// TIA Portal project "MILL" (V18)

(* hardware
DEVICE "S7-1200-Station_1"  S7-1200 Station
   slot 0: "Baugruppenträger_0"  S7-1200 Rack  Rack  V1.0
   slot 1: "MILL"  CPU 1215C DC/DC/DC  6ES7 215-1AG40-0XB0  V4.5
*)

// ===== PLC "MILL"  CPU 1215C DC/DC/DC =====

VAR_GLOBAL   // PLC tag table "Variablentabelle_1"
   "band_rein" AT %Q0.0 : Bool;   // DQa.0
   "eingang_LS" AT %I0.0 : Bool;   // DIa.0
   "bearbeitung_LS" AT %I0.1 : Bool;   // DIa.1
   "sauger_innen" AT %I0.2 : Bool;   // DIa.2
   "sauger_außen" AT %I0.3 : Bool;   // DIa.3
   "band_raus" AT %Q0.1 : Bool;   // DQa.1
   "sauger_rein" AT %Q0.2 : Bool;   // DQa.2
   "sauger_raus" AT %Q0.3 : Bool;   // DQa.3
   "sauger_unten" AT %Q0.4 : Bool;   // DQa.4
   "ventil_vakuum" AT %Q0.5 : Bool;   // DQa.5
   "kompressor" AT %Q0.6 : Bool;   // DQa.6
   "fraese" AT %Q0.7 : Bool;   // DQa.7
   "band_PWM" AT %Q1.0 : Bool;   // DQb.0
   "sauger_PWM" AT %Q1.1 : Bool;   // DQb.1
END_VAR

DATA_BLOCK "LOOP_DB"   // DB1
{ S7_Optimized_Access := 'TRUE' }
VERSION : 0.1
// stored: InstanceOfName LOOP
"LOOP"
BEGIN
END_DATA_BLOCK

FUNCTION_BLOCK "LOOP"   // FB1, SCL
{ S7_Optimized_Access := 'TRUE' }
VERSION : 0.1
   VAR
      warte : TON_TIME;
      warte_zeit : Time := T#500ms;
      warte_start : Bool;
      "step" : Int;
      pick : Bool;
      drop : Bool;
      mill : Bool;
      pick_finished : Bool;
      drop_finished : Bool;
      mill_finished : Bool;
      duration : Int := 2;
      idle : Bool;
   END_VAR
   VAR RETAIN
      modell : String := 'MILL';
   END_VAR
   VAR
      pick_failed : Bool;
      drop_failed : Bool;
      drop_aktiv : Bool;
      pick_aktiv : Bool;
      mill_aktiv : Bool;
   END_VAR
   VAR RETAIN
      zeit_prozessende : Time := T#2000MS;
      zeit_vakuumloesen : Time := T#200MS;
      zeit_saugerRunter : Time := T#700MS;
      zeit_vorFehlercheck : Time := T#2S;
   END_VAR
   VAR
      zeit_FraesPause : Time := T#1S;
   END_VAR
   VAR RETAIN
      "version" : String := '1.0';
   END_VAR
BEGIN
   #warte(IN:=#warte_start,
               PT:=#warte_zeit);

   // Stepchain MILL
   CASE #step OF
       0: // init
           #step := 1;
       1: // rdy
           #idle := TRUE;
           #pick_finished := FALSE;
           #pick_failed := FALSE;
           #drop_finished := FALSE;
           #drop_failed := FALSE;
           #mill_finished := FALSE;
           #step := 5;
       5: // Fallunterscheidung
           IF #pick THEN
               #pick_aktiv := TRUE;
               #pick := FALSE;
               #idle := FALSE;
               #step := 10;
           ELSIF #drop THEN
               #drop_aktiv := TRUE;
               #drop := FALSE;
               #idle := FALSE;
               #step := 100;
           ELSIF #mill THEN
               #mill_aktiv := TRUE;
               #mill := FALSE;
               #idle := FALSE;
               #step := 40;
           END_IF;

       200: // Ende jedes Prozesses
           "ventil_vakuum" := FALSE;
           "band_PWM" := FALSE;
           "band_raus" := FALSE;
           "band_rein" := FALSE;
           "sauger_PWM" := FALSE;
           "sauger_raus" := FALSE;
           "sauger_rein" := FALSE;
           #warte_zeit := #zeit_prozessende;
           #warte_start := TRUE;
           IF #warte.Q THEN
               #warte_start := FALSE;
               #step := 1;
           END_IF
           ;
       10: // ----------------------------------------------------- START PICK
           // sauger raus bis schalter
           "sauger_PWM" := TRUE;
           "sauger_raus":= TRUE;
           IF "sauger_außen" THEN
               "sauger_raus" := FALSE;
               #step := 20;
           END_IF;
       20: // kurz warten
           #warte_zeit := T#200ms;
           #warte_start := TRUE;
           IF #warte.Q THEN
               #warte_start := FALSE;
               #step := 21;
           END_IF;
       21: // Sauger nimmt WP auf
           "kompressor" := TRUE;
           #step := 25;
       25: // warten
           #warte_zeit := T#200ms;
           #warte_start := TRUE;
           IF #warte.Q THEN
               #warte_start := FALSE;
               #step := 22;
           END_IF;
       22: // saugerkopf nach unten
           "sauger_unten" := TRUE;
           #step := 23;
       23: // Saugerkopf aktivieren
           #warte_zeit := #zeit_saugerRunter;
           #warte_start := TRUE;
           IF #warte.Q THEN
               "ventil_vakuum" := TRUE;
               #warte_start := FALSE;
               #step := 24;
           END_IF;
       24: // saugerkopf nach oben
           #warte_zeit := T#200ms;
           #warte_start := TRUE;
           IF #warte.Q THEN
               #warte_start := FALSE;
               "sauger_unten" := FALSE;
               #step := 30;
           END_IF
           ;
       30: // Sauger fährt rein
           "sauger_rein" := TRUE;
           IF "sauger_innen" THEN
               "sauger_rein" := FALSE;
               #step := 31;
           END_IF;
       31: // saugerkopf deaktivieren
           "sauger_unten" := TRUE;
           #warte_start := TRUE;
           #warte_zeit := #zeit_saugerRunter;
           IF #warte.Q THEN
               "ventil_vakuum" := FALSE;
               #warte_start := FALSE;
               #step := 32;
           END_IF;
       32: // kompressor aus
           #warte_start := TRUE;
           #warte_zeit := #zeit_vakuumloesen;
           IF #warte.Q THEN
               "kompressor" := FALSE;
               #warte_start := FALSE;
               #step := 33;
           END_IF;
       33: // saugerkopf nach oben und aus
           "sauger_unten" := FALSE;
           #warte_start := TRUE;
           #warte_zeit := #zeit_vorFehlercheck;
           IF #warte.Q THEN
               #warte_start := FALSE;
               #step := 34;
           END_IF;
       34: // warten und fertig
           IF "eingang_LS" THEN // Fehlercheck
               #pick_failed := TRUE;
           ELSE
               #pick_finished := TRUE;
           END_IF;
           #pick_aktiv := FALSE;
           #step := 200;
               // ------------------------- END PICK
       40: // ----------------------------------------------------- START MILL
           // Power auf Band
           "band_PWM" := TRUE;
           #step := 41;
       41: // band rein wenn LS 
           "band_rein" := TRUE;
           IF NOT "bearbeitung_LS" THEN
               #step := 42;
           END_IF;
       42: // Band laufen lassen bis mittig über Fräse
           #warte_start := TRUE;
           #warte_zeit := T#200ms;
           IF #warte.Q THEN
               "band_rein" := FALSE;
               #warte_start := FALSE;
               #step := 43;
           END_IF;

           // ----------------------------------------------------------------------- AufgabenLösung
           // 
       43: // Fräsen
           "fraese" := TRUE;
           #warte_start := TRUE;
           #warte_zeit := T#1000ms * #duration;
           IF #warte.Q THEN
               #warte_start := FALSE;
               "fraese" := FALSE;
               #step := 44;
           END_IF;

       44: // warten zwischen fräsen
           #warte_start := TRUE;
           #warte_zeit := #zeit_FraesPause;
           IF #warte.Q THEN
               #warte_start := FALSE;
               #step := 45;
           END_IF;

       45: // erneutes Fräsen
           "fraese" := TRUE;
           #warte_start := TRUE;
           #warte_zeit := T#1000ms * #duration;
           IF #warte.Q THEN
               #warte_start := FALSE;
               "fraese" := FALSE;
               #step := 46;
           END_IF;



       46: // warten nach fräsen
           #warte_start := TRUE;
           #warte_zeit := T#1000ms;
           IF #warte.Q THEN
               #warte_start := FALSE;
               #step := 47;
           END_IF;

       47: // Band raus bis Eingang LS
           "band_raus" := TRUE;
           IF NOT "eingang_LS" THEN
               #step := 48;
           END_IF;
       48: // Band weiter bis mittig unter sauger
           #warte_start := TRUE;
           #warte_zeit := T#200ms;
           IF #warte.Q THEN
               "band_raus" := FALSE;
               #warte_start := FALSE;
               #step := 50;
           END_IF;
           // ----------------------------------------------------------------------- AufgabenLösung

       50: // Mill finished
           #mill_finished := TRUE;
           #mill_aktiv := FALSE;
           #step := 200;
           // ------------------------- END MILL
       100:// ----------------------------------------------------- Start DROP
           // Power auf sauger und kompressor
           "kompressor" := TRUE;
           "sauger_PWM" := TRUE;
           #step := 120;
       120: // Sauger fährt rein
           "sauger_rein" := TRUE;
           IF "sauger_innen" THEN
               "sauger_rein" := FALSE;
               #step := 101;
           END_IF;
       101: // saugerkopf nach unten
           "sauger_unten" := TRUE;
           #step := 102;
       102: // Saugerkopf aktivieren
           #warte_start := TRUE;
           #warte_zeit := #zeit_saugerRunter;
           IF #warte.Q THEN
               "ventil_vakuum" := TRUE;
               #warte_start := FALSE;
               #step := 103;
           END_IF;
       103: // saugerkopf nach oben
           #warte_zeit := T#200ms;
           #warte_start := TRUE;
           IF #warte.Q THEN
               #warte_start := FALSE;
               "sauger_unten" := FALSE;
               #step := 104;
           END_IF;
       104: // sauger raus bis schalter
           "sauger_raus" := TRUE;
           IF "sauger_außen" THEN
               "sauger_raus" := FALSE;
               #step := 105;
           END_IF;
       105: // saugerkopf nach unten
           "sauger_unten" := TRUE;
           #warte_zeit := #zeit_saugerRunter;
           #warte_start := TRUE;
           IF #warte.Q THEN
               #warte_start := FALSE;
               #step := 106;
           END_IF;
       106: // Ventil auf
           "ventil_vakuum" := FALSE;
           #warte_zeit := #zeit_vakuumloesen;
           #warte_start := TRUE;
           IF #warte.Q THEN
               #warte_start := FALSE;
               #step := 107;
           END_IF;
       107: // Kompressor aus
           "kompressor" := FALSE;
           #warte_zeit := #zeit_vakuumloesen;
           #warte_start := TRUE;
           IF #warte.Q THEN
               #warte_start := FALSE;
               #step := 108;
           END_IF;
       108: // saugerkopf nach oben
           #warte_start := TRUE;
           #warte_zeit := T#200ms;
           IF #warte.Q THEN
               "sauger_unten" := FALSE;
               #warte_start := FALSE;
               #step := 109;
           END_IF;
       109: // warten
           #warte_start := TRUE;
           #warte_zeit := T#300ms;
           IF #warte.Q THEN
               #warte_start := FALSE;
               #step := 110;
           END_IF;
       110: // reinfahren
           "sauger_rein" := TRUE;
           IF "sauger_innen" THEN
               "sauger_rein" := FALSE;
               #step := 112;
           END_IF;
       112: // drop check und ENDE
           IF NOT "eingang_LS" THEN
               #drop_failed := TRUE;
           ELSE
               #drop_finished := TRUE;
           END_IF;
           #drop_aktiv := FALSE;
           #step := 200;
           // ------------------------- END DROP
       ELSE;
   END_CASE;
END_FUNCTION_BLOCK

ORGANIZATION_BLOCK "Main"   // OB1, LAD, ProgramCycle
TITLE = "Main Program Sweep (Cycle)"
{ S7_Optimized_Access := 'TRUE' }
VERSION : 0.1
   VAR_INPUT
      Initial_Call : Bool;   // Initial call of this OB
      Remanence : Bool;   // =True, if remanent data are available
   END_VAR
BEGIN

REGION Network 1
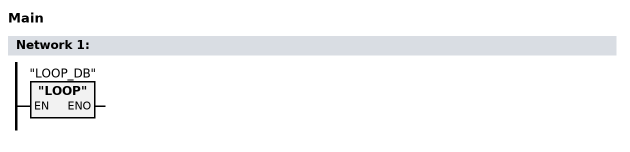
   RUNG wire#powerrail
      "LOOP_DB"()
   END_RUNG
   // the same network as SCL:
   "LOOP_DB"();   // "LOOP"
END_REGION
END_ORGANIZATION_BLOCK